PROGRAM Log_Data_Buffer
VAR
	voltage_effective : REAL;
	voltage_frequency : REAL;
	current_effective : REAL;
	current_frequency : REAL;
	power : REAL;
    fbGetCurTaskIdx  : GETCURTASKINDEX;
    ncycletime       : REAL;
	nState: INT;	
	bRecord : BOOL;
	//for generating timestamp
	fbGetSystemTime1: GetSystemTime;
	dwTimeLoDW: DWORD;
	dwTimeHiDW: DWORD;
	tFileTime: T_FILETIME;
	nTimestamp: REAL;
	
	//for insert meta data
	write_meta : BOOL;
	status_write_meta : BOOL;
	
	//for insert masur samples
	fbPLCDBCmd: FB_PLCDBCmdEvt(sNetID:= '', tTimeout:= T#19S);
	aPara: ARRAY [0..6] OF ST_ExpParameter;	
	sCmd1: STRING(255);
	sCmd2: STRING(255);
	sCmd: STRING(512); //CONCAT of sCmd1 and sCmd2
	
	//Data buffer for masur data
	aWriteSQL: ARRAY [0..19] OF BOOL;
	stData: ARRAY [0..19,0..99] OF ST_Masurdata;
	
	//buffer index and masur data variables
	nWriteBufferIndex: INT := 0;
	nWriteIndex: INT := 0;
	nSQLIndex: INT := 0;					
	bError: BOOL;
	bTableCreated: BOOL;
	bRecording: BOOL;
	nRecords: INT;
	sTableName: T_MaxString := 'masur';
	nDBID: UDINT := 1;
	index : INT := 0;
	timestampp : REAL := 0;
	
	// Eventlogger
	ipTcResult: Tc3_Database.I_TcMessage;
END_VAR

// Convert Data and get the raw data
voltage_effective := INT_TO_REAL(GVL_IO.gl_voltage_effective_raw)/65535*20; // Measured with an 
voltage_frequency := 1/(UINT_TO_REAL(GVL_IO.gl_voltage_periode_raw)/1000); //convert ms to s and get Frequency from Period

current_effective := INT_TO_REAL(GVL_IO.gl_current_effective_raw)/65535*20; // Measured with an 
current_frequency := 1/(UINT_TO_REAL(GVL_IO.gl_current_periode_raw)/1000); //convert ms to s and get Frequency from Period

fbGetCurTaskIdx();
ncycletime := _TaskInfo[fbGetCurTaskIdx.index].CycleTime/10000;

//Create timestamp
fbGetSystemTime1(timeLoDW=>dwTimeLoDW,timeHiDW=>dwTimeHiDW);
tFileTime.dwLowDateTime := dwTimeLoDW;
tFileTime.dwHighDateTime := dwTimeHiDW;	
MEMCPY(ADR(nTimestamp), ADR(tFileTime), 8);

CASE nState OF
	0://Init
		IF bRecord THEN			
			bError := FALSE;
			bRecording := FALSE;
			nRecords := 0;
			
			//sTableName := 'Magnet';//CONCAT('tbl_TestSignals_', LINT_TO_STRING(nTimestamp)); //create new tablename
						
			sCmd1 := CONCAT('INSERT INTO ', sTableName);
			sCmd2 := ' ([time2],[primary_power],[secondary_power],[phase_shift],[frequency],[flux_density],[Meta_id]) VALUES({time2},{primary_power},{secondary_power},{phase_shift},{frequency},{flux_density},{Meta_id});';
			
			CONCAT2(ADR(sCmd1), ADR(sCmd2), ADR(sCmd), SIZEOF(sCmd));
			
			aPara[0].sParaName:= 'time2'; 			aPara[0].nParaSize:= 8; 	aPara[0].eParaType:= E_ExpParameterType.Float32 ;		
			aPara[1].sParaName:= 'primary_power';	aPara[1].nParaSize:= 8;		aPara[1].eParaType:= E_ExpParameterType.Float32 ;		
			aPara[2].sParaName:= 'secondary_power';	aPara[2].nParaSize:= 8;		aPara[2].eParaType:= E_ExpParameterType.Float32 ;	
			aPara[3].sParaName:= 'phase_shift';		aPara[3].nParaSize:= 8;		aPara[3].eParaType:= E_ExpParameterType.Float32 ;
			aPara[4].sParaName:= 'frequency';		aPara[4].nParaSize:= 8;		aPara[4].eParaType:= E_ExpParameterType.Float32 ;
			aPara[5].sParaName:= 'flux_density';	aPara[5].nParaSize:= 8;		aPara[5].eParaType:= E_ExpParameterType.Float32 ;
			aPara[6].sParaName:= 'Meta_id';			aPara[6].nParaSize:= 8;		aPara[6].eParaType:= E_ExpParameterType.Int16 ;	
			nWriteBufferIndex := 0;
			nWriteIndex := 0;
			nSQLIndex := 0;	
			
			nState := 1;
		END_IF
		
	1://Idle
		IF write_meta THEN
			METH_Writemeta();
			METH_Writemeta(status => status_write_meta); //Fehlerzustand beim schreiben der Metadaten 
		END_IF
		
	2://Recording		
		bRecording := TRUE;
		
		//Fill buffer
		stData[nWriteBufferIndex, nWriteIndex].time2 := ntimestamp;
		stData[nWriteBufferIndex, nWriteIndex].primary_power := voltage_effective*current_effective;
		stData[nWriteBufferIndex, nWriteIndex].secondary_power := voltage_effective*current_effective+1;
		stData[nWriteBufferIndex, nWriteIndex].phase_shift := 1.0;
		stData[nWriteBufferIndex, nWriteIndex].frequency := 2.0;
		stData[nWriteBufferIndex, nWriteIndex].flux_density := 3.0;
		stData[nWriteBufferIndex, nWriteIndex].Meta_id := 1;
		timestampp := ncycletime * index;
		index := index + 1;
			
		//Set buffer index
		nWriteIndex := nWriteIndex + 1;		
		IF nWriteIndex = 100 THEN
			nWriteIndex := 0;
			aWriteSQL[nWriteBufferIndex]:= TRUE;
			nWriteBufferIndex := nWriteBufferIndex + 1;
			
			IF nWriteBufferIndex = 20 THEN
				nWriteBufferIndex := 0;
			END_IF 	
			
			IF aWriteSQL[nWriteBufferIndex] THEN
				nState := 255;
				RETURN;
			END_IF
		END_IF
				
		//Write buffer element (100 samples) to database
		IF aWriteSQL[nSQLIndex] THEN
			ipTcResult := fbPLCDBCmd.ipTcResult;
			IF fbPLCDBCmd.Execute(nDBID, ADR(sCmd), SIZEOF(sCmd), ADR(stData[nSQLIndex,0]), SIZEOF(stData[nSQLIndex,0]) * 100, ADR(aPara), SIZEOF(aPara)) THEN
				IF fbPLCDBCmd.bError THEN					
					nState := 255;
				ELSE
					nRecords := nRecords + 100;
					
					aWriteSQL[nSQLIndex] := FALSE;
					
					nSQLIndex := nSQLIndex + 1;
					IF nSQLIndex = 20 THEN
						nSQLIndex := 0;
					END_IF
					
					IF NOT bRecord THEN
						bRecording := FALSE;
						nState := 0;
					END_IF
				END_IF				
			END_IF
		END_IF
		
	255://Error
		bError := TRUE;
		bRecording := FALSE;
		IF NOT bRecord THEN			
			nState := 0;
		END_IF 
END_CASE

METHOD METH_Writemeta : BOOL
VAR
	stMetadata : ST_Metadata;
	fbPLCWrite : FB_PLCDBWrite(sNetID:='', tTimeout:=T#5S);
	arrColumns: ARRAY[0..32] OF STRING(255) := ['measurementname', 'carried_out', 'thickness', 'steel', 'joint_pre', 'root_face', 'opening_angel', 'edge_pre', 'welding_speed', 'laser_power', 'focal_position', 'distance_a_l', 'wire_feeding_rate', 'wire_diameter', 'wire_type', 'stickout', 'arc_dynamic', 'frequency', 'voltage_ac_power_source', 'distance_magnet_pole', 'magnet_pole_width', 'magnet_pole_type', 'core_dimension', 'very_good', 'normal', 'uniform_root_overcome', 'undercut', 'sporadic_seam_collapse', 'sporadic_dropout', 'bad', 'periodic_dropout', 'strong_seam_collapse', 'incomplite_penetration'];
END_VAR
VAR_OUTPUT
	status : BOOL;
END_VAR
// Get variables from global list form Visu Interface 
stMetadata.measurementname := GVL_Meta.measurementname;
stMetadata.carried_out := GVL_Meta.carried_out;
stMetadata.thickness := GVL_Meta.thickness;
stMetadata.steel := GVL_Meta.steel;
stMetadata.joint_pre := GVL_Meta.joint_pre;
stMetadata.root_face := GVL_Meta.root_face;
stMetadata.opening_angel := GVL_Meta.opening_angel;
stMetadata.edge_pre := GVL_Meta.edge_pre;
stMetadata.welding_speed := GVL_Meta.welding_speed;
stMetadata.laser_power := GVL_Meta.laser_power;
stMetadata.focal_position := GVL_Meta.focal_position;
stMetadata.distance_a_l := GVL_Meta.distance_a_l;
stMetadata.wire_feeding_rate := GVL_Meta.wire_feeding_rate;
stMetadata.wire_diameter := GVL_Meta.wire_diameter;
stMetadata.wire_type := GVL_Meta.wire_type;
stMetadata.stickout := GVL_Meta.stickout;
stMetadata.arc_dynamic := GVL_Meta.arc_dynamic;
stMetadata.frequency := GVL_Meta.frequency;
stMetadata.voltage_ac_power_source := GVL_Meta.voltage_ac_power_source;
stMetadata.distance_magnet_pole := GVL_Meta.distance_magnet_pole;
stMetadata.magnet_pole_width := GVL_Meta.magnet_pole_width;
stMetadata.magnet_pole_type := GVL_Meta.magnet_pole_type;
stMetadata.core_dimension := GVL_Meta.core_dimension;
stMetadata.very_good := GVL_Meta.very_good;
stMetadata.normal := GVL_Meta.normal;
stMetadata.uniform_root_overcome := GVL_Meta.uniform_root_overcome;
stMetadata.undercut := GVL_Meta.undercut;
stMetadata.sporadic_seam_collapse := GVL_Meta.sporadic_seam_collapse;
stMetadata.sporadic_dropout := GVL_Meta.sporadic_dropout;
stMetadata.bad := GVL_Meta.bad;
stMetadata.periodic_dropout := GVL_Meta.periodic_dropout;
stMetadata.strong_seam_collapse := GVL_Meta.strong_seam_collapse;
stMetadata.incomplite_penetration := GVL_Meta.incomplite_penetration;

//write struct with event to database table Meta
fbPLCWrite.WriteStruct(
	hDBID:= 1, 
	sTableName:= 'Meta', 
	pRecord:= ADR(stMetadata), 
	cbRecord:= SIZEOF(stMetadata), 
	pColumnNames:= ADR(arrColumns), 
	cbColumnNames:= SIZEOF(arrColumns));

IF fbPLCWrite.bError THEN
	status := TRUE;
ELSE
	status := FALSE;	
END_IF
END_METHOD

END_PROGRAM

(* stored: Version 1.1.0.1, ProductVersion 3.1.4024.12
   POU Log_Data_Buffer: Id {def14632-0ea6-45a1-81df-1b36ed798037}, SpecialFunc None
   Method METH_Writemeta: Id {54da36cd-3d83-45b3-b8b0-ba26b0fedece} *)
